Staubli VAL3: Axis8onPosition.pgx

public program Axis8onPosition(num x_nPos (dimensions=1), num x_nPrecent (dimensions=1), bool& x_bOK (dimensions=1))
  local num l_nNum
begin

  x_bOK=false
  call GetAxis8Pos(l_nNum,x_nPrecent)
  x_bOK=abs(l_nNum-x_nPos)<0.001

end
